FUNCTION_BLOCK Insertion //2d insertion that combines a slider (alignment) and screw (push)
VAR_INPUT //interface references to existing drives
	slider : I_PositionalDrive;
	screw : I_ContinuousDrive;
END_VAR
VAR_OUTPUT
	contact AT %I* : BOOL;
	
	active : BOOL;
	error : BOOL;
	home : BOOL;
	
	homingComplete : BOOL;
	
	sliderPos : LREAL;
END_VAR
(*
this FB encapsulates 2 drives into a generic insertion machine
both drives should be declared externally in Hardware GVL as a concrete FB
Insertion instance should be declared and called in module scope, with the drives from Hardware GVL passed in by Interface reference
*)

homingComplete := slider.HomeSet AND screw.HomeSet;

active := slider.Active OR screw.Active;
error := slider.Error OR screw.Error;
home := slider.AtHome AND screw.AtHome;

sliderPos := slider.CurrentPosition;

METHOD align : BOOL
VAR_INPUT
	targetPos : REAL;
END_VAR
slider.moveAbsolute(newTarget := targetPos);
END_METHOD

METHOD homingSequence : BOOL
VAR_INPUT
END_VAR
IF NOT slider.homeSet THEN
	slider.homingSequence();
END_IF

IF NOT screw.homeSet THEN
	screw.homingSequence();
END_IF

homingSequence := homingComplete;
END_METHOD

METHOD press : BOOL
VAR_INPUT
END_VAR
IF NOT contact THEN
	screw.moveContinuous(direction := MC_Negative_Direction);
END_IF
END_METHOD

METHOD release : BOOL
VAR_INPUT
END_VAR
screw.moveContinuous(direction := MC_Positive_Direction);
END_METHOD

METHOD reset : BOOL
VAR_INPUT
END_VAR
slider.reset();
screw.reset();
END_METHOD

METHOD stop : BOOL
VAR_INPUT
END_VAR
screw.stop();
slider.stop();
END_METHOD

METHOD toHome : BOOL
VAR_INPUT
END_VAR
slider.toHome();
screw.toHome();

toHome := slider.AtHome AND screw.AtHome;
END_METHOD

END_FUNCTION_BLOCK

(* stored: Version 1.1.0.1, ProductVersion 3.1.4024.11
   POU Insertion: Id {6fdcc75d-47a9-4376-9535-f29e878efaa0}, SpecialFunc None
   Method align: Id {faf6e411-d4af-46d2-abcb-b838ea5bab67}
   Method homingSequence: Id {ae553247-1fea-44b9-ac9e-aa5f16aca2a6}
   Method press: Id {895db015-c226-409d-96e6-d5426910ae2e}
   Method release: Id {28bb9e09-a97d-4476-bfa3-854e18353f00}
   Method reset: Id {f2128670-f949-44ac-887e-ee1dc72ef25c}
   Method stop: Id {04918701-13bc-4373-bbdc-5e7250be0092}
   Method toHome: Id {c72f4a28-e930-41f5-bda1-2377534a9b28} *)
